# B&R Automation Studio project laba11
Automation Studio 4.9

## Configuration Config1

### Task classes (Cpu.sw)
```
Cyclic#1:
  ncsdcctrl <- ncsdcctrl.prg
  Program <- Program.prg
DataObjects: Acp10sys
NcDataObjects: acp10etxen <- acp10etxen.dob, gAxis01a <- gAxis01obj.gAxis01a.dob, gAxis01i <- gAxis01obj.gAxis01i.dob, gAxis02a <- gAxis02obj.gAxis02a.dob, gAxis02i <- gAxis02obj.gAxis02i.dob
Binaries: TCData, udbdef, acp10cfg, Acp10map, iomap, arconfig, asfw, ashwac, sysconf, User, Role, ashwd
Libraries: Library, Acp10man, Acp10par, NcGlobal, Acp10sdc, Acp10_MC, brsystem, sys_lib, runtime, AsBrStr, astime, fileio, powerlnk, asieccon
```

## Logical view

Binary libraries used (declarations not repeated): operator, runtime, astime, AsIecCon, brsystem, sys_lib, AsBrStr, Acp10man, Acp10par, NcGlobal, Acp10_MC, Acp10sdc

### Package Logical/Libraries - Global libraries

### Library Logical/Libraries/Library (ANSIC)

#### Library.fun - Exported functions and function blocks
```iecst
{REDUND_ERROR} FUNCTION_BLOCK FBIntegrator (*TODO: Add your comment here*) (*$GROUP=User,$CAT=User,$GROUPICON=User.png,$CATICON=User.png*)
	VAR_INPUT
		in : REAL;
	END_VAR
	VAR_OUTPUT
		out : {REDUND_UNREPLICABLE} REAL; (*выход интегрирующего звена*)
	END_VAR
	VAR
		dt : REAL;
		oldval : {REDUND_UNREPLICABLE} REAL; (*J*)
	END_VAR
END_FUNCTION_BLOCK

{REDUND_ERROR} FUNCTION_BLOCK FBRegulator (*TODO: Add your comment here*) (*$GROUP=User,$CAT=User,$GROUPICON=User.png,$CATICON=User.png*)
	VAR
		dt : REAL;
		e : REAL; (*рассогласование между задающим воздействием и реальной скоростью вращения вала ДПТ [об/мин]*)
		u : REAL; (*напряжение, подаваемое на вход ДПТ [В]*)
		k_p : REAL; (*пропорциональный коэффициент регулятора*)
		k_i : REAL; (*интегральный коэффициент регулятора*)
		integrator : FBIntegrator; (*интегратор *)
		iyOld : REAL; (*хранение предыдущего значения схемы противонакопления*)
		max_abs_value : REAL; (*граница блока ограничения [В]*)
	END_VAR
END_FUNCTION_BLOCK

{REDUND_ERROR} FUNCTION_BLOCK FBMotor (*TODO: Add your comment here*) (*$GROUP=User,$CAT=User,$GROUPICON=User.png,$CATICON=User.png*)
	VAR_INPUT
		u : REAL; (*входное напряжение [В]*)
		Tm : REAL; (*частота вращения [об/мин]*)
	END_VAR
	VAR_OUTPUT
		w : REAL; (*интегратор *)
		phi : REAL; (*электромеханическая постоянная времени [с]*)
	END_VAR
	VAR
		dt : REAL;
		ke : REAL; (*положение [рад]*)
		integrator : FBIntegrator; (*постоянная ЭДС двигателя [В•мин/об]*)
		integrator1 : FBIntegrator;
	END_VAR
END_FUNCTION_BLOCK

{REDUND_ERROR} FUNCTION_BLOCK FBMotor1 (*TODO: Add your comment here*) (*$GROUP=User,$CAT=User,$GROUPICON=User.png,$CATICON=User.png*)
	VAR
		dt : REAL;
	END_VAR
	VAR_INPUT
		u : REAL; (*входное напряжение [В]*)
		Tm : REAL; (*частота вращения [об/мин]*)
	END_VAR
	VAR_OUTPUT
		w : REAL; (*интегратор *)
		phi : REAL; (*электромеханическая постоянная времени [с]*)
	END_VAR
	VAR
		ke : REAL; (*положение [рад]*)
		integrator : FBIntegrator; (*постоянная ЭДС двигателя [В•мин/об]*)
		integrator1 : FBIntegrator;
	END_VAR
END_FUNCTION_BLOCK
```

#### FBIntegrator.c
```c
#include <bur/plctypes.h>
#ifdef __cplusplus
	extern "C"
	{
#endif
	#include "Library.h"
#ifdef __cplusplus
	};
#endif
/* TODO: Add your comment here */
void FBIntegrator(struct FBIntegrator* inst)
{
	inst->out = inst->oldval + ((inst->in) * inst->dt);
	inst->oldval = inst->out;
}
```

#### FBRegulator.c
```c
#include <bur/plctypes.h>
#ifdef __cplusplus
	extern "C"
	{
#endif
	#include "Library.h"
#ifdef __cplusplus
	};
#endif
/* TODO: Add your comment here */
void FBRegulator(struct FBRegulator* inst)
{
	REAL temp;
	temp = inst->e * inst->k_i * inst->dt;
	temp+=inst->iyOld;
	inst->integrator.in = temp;
	inst->integrator.dt = inst->dt;
	FBIntegrator(&inst->integrator);

	if (inst->e * inst->k_p > inst->max_abs_value)
	{
		temp = inst->integrator.out + inst->max_abs_value;
	}
	if (inst->e * inst->k_p < inst->max_abs_value)
	{
		temp = inst->integrator.out + inst->e * inst->k_p;
	}
	if (temp > inst->max_abs_value)
	{
		inst->u = inst->max_abs_value;
		inst->iyOld = temp - inst->max_abs_value;
	}
	else
	{
		inst->u = temp;
		inst->iyOld = 0;
	}
}
```

#### FBMotor.c
```c
#include <bur/plctypes.h>
#ifdef __cplusplus
	extern "C"
	{
#endif
	#include "Library.h"
#ifdef __cplusplus
	};
#endif
/* TODO: Add your comment here */
void FBMotor(struct FBMotor* inst)
{
	REAL temp;
	temp = inst->u / inst->ke;
	temp = temp - inst->w;
	temp = temp * inst->dt / inst->Tm;
	inst->integrator.in = temp;
	inst->integrator.dt = inst->dt;
	inst->integrator1.dt = inst->dt;
	FBIntegrator(&inst->integrator);
	temp = inst->integrator.out;
	inst->w = temp;
	temp = inst->w;
	inst->integrator1.in = temp;
	FBIntegrator(&inst->integrator1);
	inst->phi = inst->integrator1.out;
	/*TODO: Add your code here*/
}
```

#### FBMotor1.c
```c
#include <bur/plctypes.h>
#ifdef __cplusplus
	extern "C"
	{
#endif
	#include "Library.h"
#ifdef __cplusplus
	};
#endif
/* TODO: Add your comment here */
void FBMotor1(struct FBMotor1* inst)
{
	REAL temp;
	temp = inst->u / inst->ke;
	temp = temp - inst->w;
	temp = temp * inst->dt / inst->Tm;
	inst->integrator.in = temp;
	inst->integrator.dt = inst->dt;
	inst->integrator1.dt = inst->dt;
	FBIntegrator(&inst->integrator);
	temp = inst->integrator.out;
	inst->w = temp;
	temp = inst->w;
	inst->integrator1.in = temp;
	FBIntegrator(&inst->integrator1);
	inst->phi = inst->integrator1.out;
	/*TODO: Add your code here*/
}
```

### Program Logical/Program (ANSIC)

#### Variables.var
```iecst
VAR
	fb_motor : FBMotor;
	Speed : REAL;
	fb_reg : FBRegulator;
	timecount : REAL;
	Enable : BOOL;
	t : REAL;
	ResW : REAL;
	ResPhi : REAL;
	fb_motor1 : FBMotor1;
	temp : REAL;
END_VAR
```

#### Main.c
```c
#include <bur/plctypes.h>
#include <math.h>

#ifdef _DEFAULT_INCLUDES
	#include <AsDefault.h>
#endif

void _INIT ProgramInit(void)
{
	t = 0;
	fb_reg.k_i = 0.16;
	fb_reg.k_p = 0.0064;
	fb_motor.dt = 0.002;
	fb_motor.Tm = 0.04;
	fb_motor.ke = 0.002;
	fb_reg.dt = 0.002;
	fb_reg.e = 0;
	fb_reg.max_abs_value = 300;
	fb_motor1.u = 0;
	fb_motor1.dt = 0.002;
	fb_motor1.Tm = 0.01;
	fb_motor1.ke = 0.2;
	Enable  = 1;

}

void _CYCLIC ProgramCyclic(void)
{
	if (Enable == 1)
	{
		Speed = 100;
	}
	if (Enable == 0)
	{
		Speed = 0;
	}
	t = t + 0.002;
	fb_reg.e = Speed - fb_motor.w;
	FBRegulator(&fb_reg);
	fb_motor.u = fb_reg.u;
	FBMotor(&fb_motor);
	ResW = fb_motor.w;
	ResPhi = fb_motor.phi;
	FBMotor1(&fb_motor1);
	fb_motor1.u = Speed - fb_motor1.w;
	if ((t > 2)){
		Enable = !Enable;
		t = 0;
	}

}

void _EXIT ProgramExit(void)
{

}
```

Listed in the project but not available here: Logical/Global.typ, Logical/Global.var, Logical/Libraries/Library/Types.typ, Logical/Libraries/Library/Constants.var, Logical/ncsdcctrl, Logical/acp10etxen, Logical/gAxis01obj, Logical/gAxis02obj
